# EPICS autosave request: mcaApp/Db/icb_tca_settings.req
# FILE... icb_tca_settings.req
# USAGE.. icb_tca.db fields autosave'd.
$(P)$(TCA)POLARITY
$(P)$(TCA)THRESHOLD
$(P)$(TCA)SCA_ENABLE
$(P)$(TCA)SCA1_GATE
$(P)$(TCA)SCA2_GATE
$(P)$(TCA)SCA3_GATE
$(P)$(TCA)TCA_SELECT
$(P)$(TCA)PUR_ENABLE
$(P)$(TCA)SCA1_PUR
$(P)$(TCA)SCA2_PUR
$(P)$(TCA)SCA3_PUR
$(P)$(TCA)PUR_AMP
$(P)$(TCA)SCA1_LOW
$(P)$(TCA)SCA1_HI
$(P)$(TCA)SCA2_LOW
$(P)$(TCA)SCA2_HI
$(P)$(TCA)SCA3_LOW
$(P)$(TCA)SCA3_HI
$(P)$(TCA)ROI_SCA_ENABLE
$(P)$(TCA)SCA_CAL
